Staubli VAL3: DecToHex.pgx

public program DecToHex(num x_nDecimal, string& x_sHex)
  local num l_nRest
  local num l_nDecimal
  local num l_nIndex
begin

  //only integers allowed!
  l_nDecimal = round(x_nDecimal)
  resize(sDecHexBuff, 1, 1)

  while l_nDecimal != 0

    l_nRest = l_nDecimal % 16
    sDecHexBuff[size(sDecHexBuff)-1] = sDec2HexSymbols[l_nRest]
    append(sDecHexBuff)
    l_nDecimal = roundDown(l_nDecimal/16)

  endWhile

  x_sHex = ""
  for l_nIndex = size(sDecHexBuff)-1 to 0 step-1
    x_sHex = x_sHex + sDecHexBuff[l_nIndex]
  endFor


end
